FUNCTION_BLOCK Test_ReadWriteBySymbolName EXTENDS T_UnitTestBase
VAR
    AdsReadWriteBySymbolName : T_AdsReadWriteBySymbolName;
    TestInteger : TInteger;
    ReadWriteResult : INT;    
    ScanCount : DINT;
    State: INT;
END_VAR

CASE State OF
    0:
        TestInteger.Init(1111);
        ReadWriteResult := 0;
        ScanCount := 0;
    
        AdsReadWriteBySymbolName.Execute(
            AmsNetId:= '', 
            Port:= Constants.PortNo, 
            SymbolName:= 'PB_TestRunner.Test_ReadWriteBySymbolName.TestInteger#Inc', 
            ReadDataAddress:= ADR(ReadWriteResult), 
            ReadDataLength:= SIZEOF(ReadWriteResult), 
            WriteDataAddress:= 0, 
            WriteDataLength:= 0, 
            KeepSymbolHandle:= FALSE);


        State := 10;
        
    10:
        ScanCount := ScanCount + 1;
        IF NOT AdsReadWriteBySymbolName.Execution.Busy THEN
            State := 20;    
		END_IF
        
    20:
        Assertion.AssertEquals_INT(
            Expected     := 1112,
            Actual       := ReadWriteResult,
            Variablename := 'ReadWriteResult'); 
 
        TestFinished();
        State := 0;
END_CASE

AdsReadWriteBySymbolName();

END_FUNCTION_BLOCK

(* stored: Version 1.1.0.1, ProductVersion 3.1.4024.4
   POU Test_ReadWriteBySymbolName: Id {46315f3c-bda6-0e0c-3cc9-f95106c4e9c3}, SpecialFunc None *)
